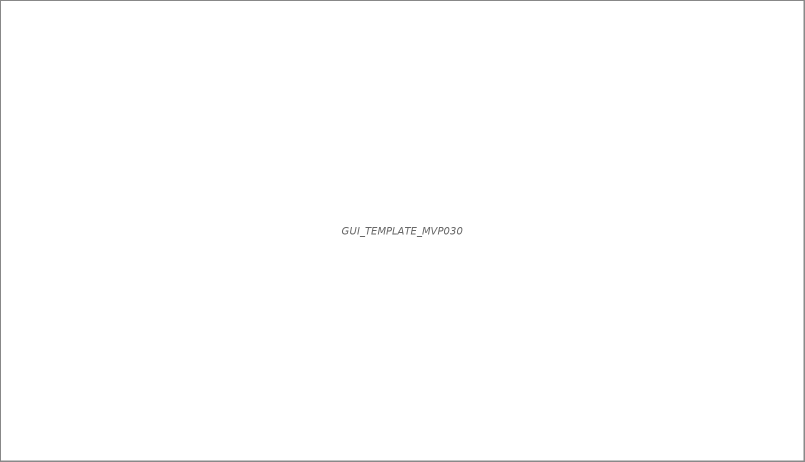
VISUALIZATION GUI_MVP030_EVAC_PDS  // 805x462
    Frame (0,0 805x462)
        shows GUI_TEMPLATE_MVP030(m_Instance := MAIN.evac_pds.rp, m_bEnable := MAIN.evac_pds.ctrl.bEnable_RP)
END_VISUALIZATION

(* stored: Version 1.1.0.1, ProductVersion 3.1.4024.9
   Visu GUI_MVP030_EVAC_PDS: Id {41387eb1-d541-4ee6-8c9d-558b7d493b87} *)
